INTERFACE ITF_Sender EXTENDS __System.IQueryInterface

PROPERTY SendData : ST_CommunicationMetaData
GET
END_GET
END_PROPERTY

END_INTERFACE

(* stored: Version 1.1.0.1, ProductVersion 3.1.4024.15
   Itf ITF_Sender: Id {f4a66d46-a96f-4600-9bdf-2da59ac2218f}
   Property SendData: Id {c66ebad0-9ef6-41b4-aa9b-204d70c67f9e}
   Get Get: Id {67c79e9a-daf0-46d3-b7eb-e2a36a9cec8b} *)
